(* PLC project SafeLOGIC, BrAutomation SafeDESIGNER  5.24.1.0 *)
(* stored: companyURL http://www.br-automation.com, creationDateTime Sun Oct 26 13:20:31 2025 *)

PROGRAM Main

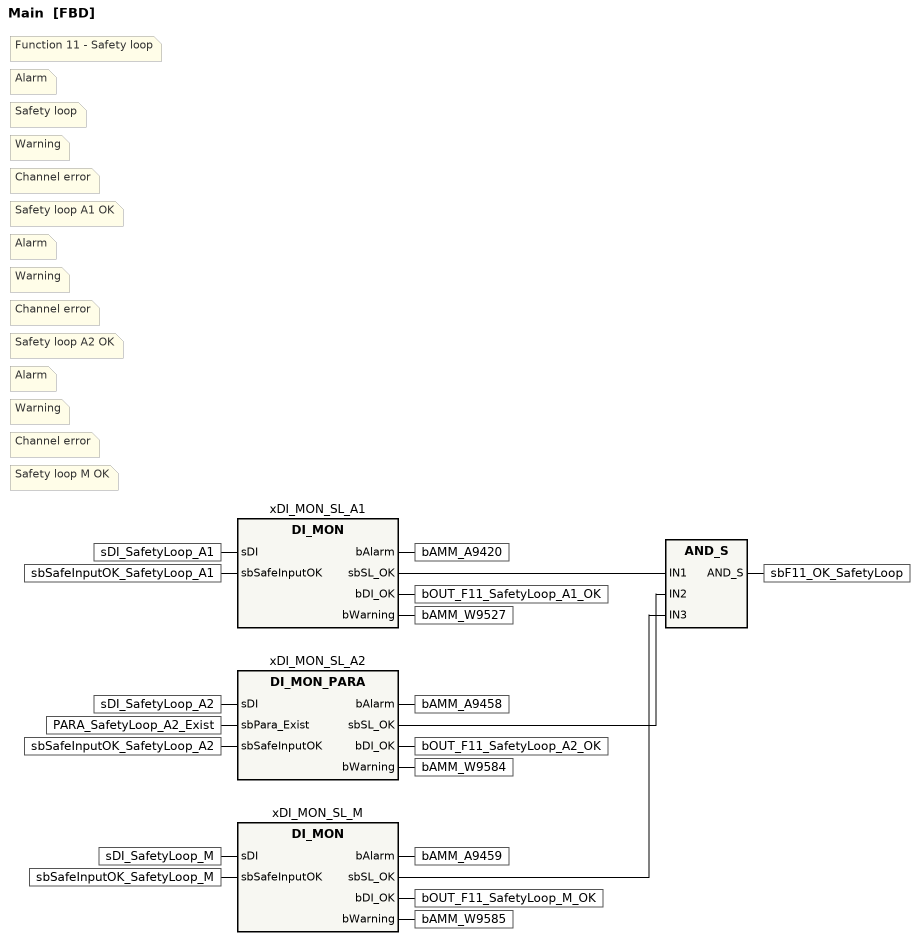
(* FBD diagram, written out as Structured Text *)
(* Function 11 - Safety loop *)
(* Alarm *)
xDI_MON_SL_A1(sDI := sDI_SafetyLoop_A1, sbSafeInputOK := sbSafeInputOK_SafetyLoop_A1);
bAMM_A9420 := xDI_MON_SL_A1.bAlarm;
(* Safety loop A1 OK *)
(* Channel error *)
(* Warning *)
bAMM_W9527 := xDI_MON_SL_A1.bWarning;
bOUT_F11_SafetyLoop_A1_OK := xDI_MON_SL_A1.bDI_OK;
(* Alarm *)
xDI_MON_SL_A2(sDI := sDI_SafetyLoop_A2, sbPara_Exist := PARA_SafetyLoop_A2_Exist, sbSafeInputOK := sbSafeInputOK_SafetyLoop_A2);
bAMM_A9458 := xDI_MON_SL_A2.bAlarm;
(* Safety loop A2 OK *)
(* Channel error *)
(* Warning *)
bAMM_W9584 := xDI_MON_SL_A2.bWarning;
bOUT_F11_SafetyLoop_A2_OK := xDI_MON_SL_A2.bDI_OK;
(* Alarm *)
xDI_MON_SL_M(sDI := sDI_SafetyLoop_M, sbSafeInputOK := sbSafeInputOK_SafetyLoop_M);
bAMM_A9459 := xDI_MON_SL_M.bAlarm;
(* Safety loop M OK *)
(* Channel error *)
(* Warning *)
bOUT_F11_SafetyLoop_M_OK := xDI_MON_SL_M.bDI_OK;
(* Safety loop *)
sbF11_OK_SafetyLoop := AND_S(xDI_MON_SL_A1.sbSL_OK, xDI_MON_SL_A2.sbSL_OK, xDI_MON_SL_M.sbSL_OK);
bAMM_W9585 := xDI_MON_SL_M.bWarning;
END_PROGRAM
